// TwinCAT 3 PLC project TcGeodetic
// Title: TcGeodetic
// Company: Burks Engineering
// Author: Andrew Burks
// ProjectVersion: 0.2.3
// Description: Geodetic transformation library
// ProgramVersion: 3.1.4023.0
// libraries:
//   Tc2_Standard, * (Beckhoff Automation GmbH)
//   Tc2_System, * (Beckhoff Automation GmbH)
//   TcMatrix, * (Burks Engineering)
//   TcTransform, * (Burks Engineering)
// project tree:
//   GVLs/ GeoEllipsoids.TcGVL
//   POUs/ GeoEllipsoid.TcPOU, GeoPose.TcPOU, GeoPosition.TcPOU
//   Version/ Global_Version.TcGVL

// ---- GVLs/GeoEllipsoids.TcGVL
{attribute 'qualified_only'}
VAR_GLOBAL
	WGS84 : GeoEllipsoid('WGS-84', 6378137.0, 1.0 / 298.257223563);
	GRS80 : GeoEllipsoid('GRS-80', 6378137.0, 1.0 / 298.257222101);
	PZ90 :  GeoEllipsoid('PZ-90' , 6378136.0, 1.0 / 298.257839303);
END_VAR

// ---- Version/Global_Version.TcGVL
{attribute 'TcGenerated'}
{attribute 'no-analysis'}
{attribute 'linkalways'}
// This function has been automatically generated from the project information.
VAR_GLOBAL CONSTANT
	{attribute 'const_non_replaced'}
	stLibVersion_TcGeodetic : ST_LibVersion := (iMajor := 0, iMinor := 2, iBuild := 3, iRevision := 0, nFlags := 0, sVersion := '0.2.3');
END_VAR

// ---- POUs/GeoEllipsoid.TcPOU
(*
Geodetic Ellipsoid
----------------

Overview
================

Represents a geodetic reference ellipsoid (but not a geodetic datum). Contains functions for transitioning between latitude/longitude and XYZ coordinates.

To access standard ellipsoids use the GVL 'GeoEllipsoids'.	They cannot be copied, but you can use REFERENCE TO types to keep a shorthand copy somewhere.

.. note:: When creating an instance of this FB you *must* provide the name, semimajor axis, and flattening due to the use of FB_init parameters.
*)
{attribute 'no_assign'}
FUNCTION_BLOCK GeoEllipsoid
VAR_INPUT
END_VAR
VAR_OUTPUT
END_VAR
VAR
	Name_ : T_MaxString;
	SemiMajorAxis_ : LREAL;
	Flattening_ : LREAL;
END_VAR

METHOD FB_init : BOOL
VAR_INPUT
	bInitRetains : BOOL; // if TRUE, the retain variables are initialized (warm start / cold start)
	bInCopyCode : BOOL;  // if TRUE, the instance afterwards gets moved into the copy code (online change)
	
	eName : T_MaxString;
	eSemiMajorAxis : LREAL;//meters
	eFlattening : LREAL;//very small number
END_VAR
Name_ := eName;
SemiMajorAxis_ := eSemiMajorAxis;
Flattening_ := eFlattening;
END_METHOD

PROPERTY PUBLIC Flattening : LREAL
GET
Flattening := Flattening_;
END_GET
END_PROPERTY

METHOD PUBLIC GetCartesianFromGeodetic : Vector3
VAR_INPUT
	P : GeoPosition;
END_VAR
VAR
	N : LREAL;
END_VAR
N := GetNormalRadiusOfCurvature(P.LatitudeRad);

GetCartesianFromGeodetic.X := (N + P.Elevation) * COS(P.LatitudeRad) * COS(P.LongitudeRad);
GetCartesianFromGeodetic.Y := (N + P.Elevation) * COS(P.LatitudeRad) * SIN(P.LongitudeRad);
GetCartesianFromGeodetic.Z := ((1.0 - GetEccentricitySquared())*N + P.Elevation) * SIN(P.LatitudeRad);
END_METHOD

METHOD PROTECTED GetEccentricitySquared : LREAL
VAR_INPUT
END_VAR
GetEccentricitySquared := (2.0-Flattening)*Flattening;
END_METHOD

METHOD PROTECTED GetGeocentricLatitude : LREAL//radians
VAR_INPUT
	GeodeticLatitude : LREAL;//radians
END_VAR
GetGeocentricLatitude := ATAN((1-Flattening_) * (1-Flattening_)*TAN(GeodeticLatitude));
END_METHOD

METHOD PUBLIC GetGeodeticFromCartesian : GeoPosition
VAR_INPUT
	V : Vector3;
END_VAR
VAR
	RadLatitude_2 : LREAL;// 		'Q^2' 		from paper
	Magnitude_2 : LREAL;// 			'r^2' 		from paper
	Eccentricity_2 : LREAL;// 		'E^2' 		from paper
	AdjustedMag_2 : LREAL;// 		'r^2 - E^2' from paper
	SemiMinorConfocal_2 : LREAL;// 	'u^2' 		from paper
	SemiMajorConfocal_2 : LREAL;// 	'u^2' + E^2 from paper
	TanGeocentricLatitude : LREAL;// tan(beta) 	from paper
	GeocentricLatitude : LREAL;//   'beta' 		from paper
	AxialElevation : LREAL;
	RadialElevation : LREAL;
END_VAR
//stolen from : http://ir.lib.ncku.edu.tw/bitstream/987654321/39750/1/3011200501001.pdf
//error is <1mm for anything within 100km of the surface of the earth

RadLatitude_2 := V.X*V.X + V.Y*V.Y;
Magnitude_2 := RadLatitude_2 + V.Z* V.Z;

//right at pole longitude is indetermiante
IF RadLatitude_2 = 0 THEN
	GetGeodeticFromCartesian.LongitudeRad := 0;
ELSE
	GetGeodeticFromCartesian.LongitudeRad := atan2(V.Y,V.X);//eq 4c from paper
END_IF

//too close to poles for stuff to work well
IF RadLatitude_2 < (SemiMajorAxis * SemiMinorAxis * 1E-32) THEN
	//center of earth...angles dont even matter anymore
	IF V.Z = 0 THEN
		GetGeodeticFromCartesian.LatitudeRad := 0;
		GetGeodeticFromCartesian.Elevation := Magnitude_2;
	ELSE
		GetGeodeticFromCartesian.LatitudeRad := PI /2 * V.Z / ABS(V.Z);
		GetGeodeticFromCartesian.Elevation := ABS(V.Z) - SemiMinorAxis;
	END_IF;
ELSE
	Eccentricity_2 := SemiMajorAxis*SemiMajorAxis - SemiMinorAxis * SemiMinorAxis;
	AdjustedMag_2 := Magnitude_2 - Eccentricity_2;
	SemiMinorConfocal_2 := 0.5*AdjustedMag_2 + 0.5*SQRT(EXPT(AdjustedMag_2,2) + 4*Eccentricity_2*V.Z*V.Z); //eq 4a from paper
	SemiMajorConfocal_2 := SemiMinorConfocal_2 + Eccentricity_2;
	IF SQRT(SemiMinorConfocal_2) / SQRT(SemiMajorConfocal_2) < 10E-10 THEN
		//avoid divide by near zero when confocal is nearly flat and assumption of geocentric latidude equivalence atan(confocal) ~= atan(ellipsoid) stops being true
		IF V.Z = 0 THEN
			GeocentricLatitude := 0;
		ELSE
			GeocentricLatitude := PI/2 * V.Z/ABS(V.Z);
		END_IF;
		GetGeodeticFromCartesian.LatitudeRad := GeocentricLatitude;
	ELSE
		TanGeocentricLatitude := (SQRT(SemiMajorConfocal_2) * V.Z) / (SQRT(SemiMinorConfocal_2)*SQRT(RadLatitude_2));
		GeocentricLatitude := ATAN(TanGeocentricLatitude); //eq 6 from paper
		GetGeodeticFromCartesian.LatitudeRad := ATAN(SemiMajorAxis / SemiMinorAxis * TanGeocentricLatitude);
	END_IF;
	
	AxialElevation := V.Z - SemiMinorAxis*SIN(GeocentricLatitude);
	RadialElevation := SQRT(RadLatitude_2) - SemiMajorAxis*COS(GeocentricLatitude);
	
	GetGeodeticFromCartesian.Elevation := SQRT(AxialElevation*AxialElevation + RadialElevation*RadialElevation); //eq 7 from paper
	IF AxialElevation < 0 AND RadialElevation < 0 THEN
		GetGeodeticFromCartesian.Elevation := -1 * GetGeodeticFromCartesian.Elevation;
	END_IF

END_IF
END_METHOD

METHOD PROTECTED GetNormalRadiusOfCurvature : LREAL
VAR_INPUT
	lat : LREAL;//radians
END_VAR
VAR
	acosf : LREAL;
	bcosf : LREAL;
	den : LREAL;
END_VAR
acosf := SemiMajorAxis * COS(lat);
bcosf := GetSemiMinorAxis() * SIN(lat);
den := SQRT(acosf*acosf + bcosf*bcosf);
IF den = 0 THEN
	GetNormalRadiusOfCurvature := 0;
	ADSLOGSTR(ADSLOG_MSGTYPE_WARN,'GeodeticPosition::GetNormalRadiusOfCurvature Divide By Zero attempt in reference ellipsoid %s',Name);
	RETURN;
END_IF
GetNormalRadiusOfCurvature := SemiMajorAxis*SemiMajorAxis/den;
END_METHOD

METHOD PROTECTED GetSemiMinorAxis : LREAL
VAR_INPUT
END_VAR
GetSemiMinorAxis := SemiMajorAxis * (1-Flattening);
END_METHOD

METHOD PUBLIC GetTangentEnuRotation : RMatrix
VAR_INPUT
	P : GeoPosition;
END_VAR
VAR
	R_ENU : RMatrix;
	R_Lon : Rmatrix;
	R_Lat : Rmatrix;
	V : Vector3;
END_VAR
GetTangentEnuRotation := GetTangentXyuRotation(P,0.0);
RETURN;

//ECEF has X as 'up',   y as 'east',  Z as 'north' as lat=lon=0, translated to surface
//ENU  has X as 'east', y as 'north', z as 'up'
//therefore, the base rotation (ignoring lat/lon changes) should be: (projecting ENU unit vecotrs onto ECEF CS)
// [  0   0   1
//    1   0   0
//    0   1   0   ]

GetTangentEnuRotation.FillTrapezoidal(0,0,0);
GetTangentEnuRotation.SetRC(1,0,1);
GetTangentEnuRotation.SetRC(2,1,1);
GetTangentEnuRotation.SetRC(0,2,1);


R_Lon.SetFromAngle(P.LongitudeRad,Dimension.Z);//positive intrinsic rotation around ECEF Z
R_Lat.SetFromAngle(-1*P.LatitudeRad,Dimension.Y);//negative instrinsic rotation around rotated ECEF Y

GetTangentEnuRotation.RotateBy(R_Lat);
GetTangentEnuRotation.RotateBy(R_Lon);
END_METHOD

METHOD PUBLIC GetTangentEnuTransform : HMatrix
VAR_INPUT
	P : GeoPosition;
END_VAR
VAR
	R_ENU : RMatrix;
	R_Lon : Rmatrix;
	R_Lat : Rmatrix;
	V : Vector3;
END_VAR
V := GetCartesianFromGeodetic(P);
GetTangentEnuTransform.SetFromComponents(GetTangentEnuRotation(P),V);
END_METHOD

METHOD PUBLIC GetTangentXyuRotation : RMatrix
VAR_INPUT
	P : GeoPosition;
	Angle : LREAL;//radians of extra angle around the 'up' vector, from ENU
END_VAR
VAR
	R_ENU : RMatrix;
	R_Lon : Rmatrix;
	R_Lat : Rmatrix;
	RHeading : RMatrix;
	V : Vector3;
END_VAR
//ECEF has X as 'up',   y as 'east',  Z as 'north' as lat=lon=0, translated to surface
//ENU  has X as 'east', y as 'north', z as 'up'
//therefore, the base rotation (ignoring lat/lon changes) should be: (projecting ENU unit vecotrs onto ECEF CS)
// [  0   0   1
//    1   0   0
//    0   1   0   ]

GetTangentXyuRotation.SetFromAngle(Angle,Dimension.Z);

R_ENU.FillTrapezoidal(0,0,0);
R_ENU.SetRC(1,0,1);
R_ENU.SetRC(2,1,1);
R_ENU.SetRC(0,2,1);

R_Lon.SetFromAngle(P.LongitudeRad,Dimension.Z);//positive intrinsic rotation around ECEF Z
R_Lat.SetFromAngle(-1*P.LatitudeRad,Dimension.Y);//negative instrinsic rotation around rotated ECEF Y

GetTangentXyuRotation.RotateBy(R_ENU);
GetTangentXyuRotation.RotateBy(R_Lat);
GetTangentXyuRotation.RotateBy(R_Lon);
END_METHOD

METHOD PUBLIC GetTangentXyuTransform : HMatrix
VAR_INPUT
	P : GeoPosition;
	Angle : LREAL;//radians of extra normal rotation
END_VAR
VAR
	R_ENU : RMatrix;
	R_Lon : Rmatrix;
	R_Lat : Rmatrix;
	V : Vector3;
END_VAR
V := GetCartesianFromGeodetic(P);
GetTangentXyuTransform.SetFromComponents(GetTangentXyuRotation(P,Angle),V);
END_METHOD

PROPERTY PUBLIC Name : T_MaxString
GET
Name := Name_;
END_GET
END_PROPERTY

//meters
PROPERTY PUBLIC SemiMajorAxis : LREAL
GET
SemiMajorAxis := SemiMajorAxis_;
END_GET
END_PROPERTY

PROPERTY PUBLIC SemiMinorAxis : LREAL
GET
SemiMinorAxis := SemiMajorAxis*(1-Flattening);
END_GET
END_PROPERTY

END_FUNCTION_BLOCK

// ---- POUs/GeoPosition.TcPOU
(*
Geographic Position
----------------

Overview
================

Represents a geodetic (or geocentric) position with latitude, longitude, and elevation (above the ellipsoid).
*)
FUNCTION_BLOCK GeoPosition
VAR_INPUT
END_VAR
VAR_OUTPUT
END_VAR
VAR
	Latitude_  : LREAL;//radians north of equator
	Longitude_ : LREAL;//radians east of meridian
	Elevation_ : LREAL;//m above ellipsoid
END_VAR

METHOD PUBLIC Clear
VAR_INPUT
END_VAR
Latitude_ := 0;
Longitude_ := 0;
Elevation_ := 0;
END_METHOD

METHOD PUBLIC CopyFrom
VAR_INPUT
	P : GeoPosition;
END_VAR
Latitude_ := P.LatitudeRad;
Longitude_ := P.LongitudeRad;
Elevation_ := P.Elevation;
END_METHOD

PROPERTY PUBLIC Elevation : LREAL
GET
Elevation := Elevation_;
END_GET
SET
Elevation_ := Elevation;
END_SET
END_PROPERTY

METHOD PUBLIC GetCartesianPosition : Vector3
VAR_INPUT
	Ref : REFERENCE TO GeoEllipsoid := GeoEllipsoids.WGS84;
END_VAR
IF NOT(__ISVALIDREF(Ref)) THEN
	GetCartesianPosition := GeoEllipsoids.WGS84.GetCartesianFromGeodetic(THIS^);
ELSE
	GetCartesianPosition := Ref.GetCartesianFromGeodetic(THIS^);
END_IF;
END_METHOD

//Gets the relative position of the supplied GeoPosition, considering this GeoPosition as an ENU tangent reference frame
METHOD PUBLIC GetRelativePosition : Vector3
VAR_INPUT
	P : GeoPosition;
	Ref : REFERENCE TO GeoEllipsoid := GeoEllipsoids.WGS84;
END_VAR
VAR
	EnuInEcef : HMatrix;
END_VAR
EnuInEcef := GetTangentEnuTransform(Ref);
GetRelativePosition := EnuInEcef.GetTransformedVector3Reverse(P.GetCartesianPosition(Ref));
END_METHOD

METHOD PUBLIC GetTangentEnuPose : GeoPose
VAR_INPUT
	Ref : REFERENCE TO GeoEllipsoid := GeoEllipsoids.WGS84;
END_VAR
GetTangentEnuPose.SetFromEcefTransformation(GetTangentEnuTransform(Ref),Ref);
END_METHOD

METHOD PUBLIC GetTangentEnuRotation : RMatrix
VAR_INPUT
	Ref : REFERENCE TO GeoEllipsoid := GeoEllipsoids.WGS84;
END_VAR
IF NOT(__ISVALIDREF(Ref)) THEN
	GetTangentEnuRotation := GeoEllipsoids.WGS84.GetTangentEnurotation(THIS^);
ELSE
	GetTangentEnuRotation := Ref.GetTangentEnurotation(THIS^);
END_IF
END_METHOD

METHOD PUBLIC GetTangentEnuTransform : HMatrix
VAR_INPUT
	Ref : REFERENCE TO GeoEllipsoid := GeoEllipsoids.WGS84;
END_VAR
IF NOT(__ISVALIDREF(Ref)) THEN
	GetTangentEnuTransform := GeoEllipsoids.WGS84.GetTangentEnuTransform(THIS^);
ELSE
	GetTangentEnuTransform := Ref.GetTangentEnuTransform(THIS^);
END_IF
END_METHOD

METHOD PUBLIC IsEqual : BOOL
VAR_INPUT
	P : REFERENCE TO GeoPosition;
END_VAR
IsEqual := IsNearlyEqual(P,0.0,0.0);
END_METHOD

METHOD PUBLIC IsNearlyEqual : BOOL
VAR_INPUT
	P : REFERENCE TO GeoPosition;
	PrecisionLatLon : LREAL;//radians
	PrecisionElevation : LREAL;//meters
END_VAR
IsNearlyEqual := ABS(P.LatitudeRad 		- LatitudeRad) 	<= PrecisionLatLon
             AND ABS(P.LongitudeRad 	- LongitudeRad) <= PrecisionLatLon
             AND ABS(P.Elevation 		- Elevation)	<= PrecisionElevation;
END_METHOD

PROPERTY PUBLIC LatitudeDeg : LREAL
GET
LatitudeDeg := 180.0 * Latitude_ /PI;
END_GET
SET
Latitude_ := PI * LatitudeDeg / 180.0;
END_SET
END_PROPERTY

PROPERTY PUBLIC LatitudeRad : LREAL
GET
LatitudeRad := Latitude_;
END_GET
SET
Latitude_ := LatitudeRad;
END_SET
END_PROPERTY

PROPERTY PUBLIC LongitudeDeg : LREAL
GET
LongitudeDeg := 180.0 * Longitude_ /PI;
END_GET
SET
Longitude_ := PI * LongitudeDeg / 180.0;
END_SET
END_PROPERTY

PROPERTY PUBLIC LongitudeRad : LREAL
GET
LongitudeRad := Longitude_;
END_GET
SET
Longitude_ := LongitudeRad;
END_SET
END_PROPERTY

METHOD PUBLIC SetFromCartesianPosition
VAR_INPUT
	V : Vector3;
	Ref : REFERENCE TO GeoEllipsoid;
END_VAR
VAR
	P : GeoPosition;
END_VAR
IF NOT(__ISVALIDREF(Ref)) THEN
	P := GeoEllipsoids.WGS84.GetGeodeticFromCartesian(V);
ELSE
	P := Ref.GetGeodeticFromCartesian(V);
END_IF
CopyFrom(P);
END_METHOD

METHOD PUBLIC SetFromComponentsDeg
VAR_INPUT
	Lat : LREAL;
	Lon : LREAL;
	El : LREAL;
END_VAR
LatitudeDeg := Lat;
LongitudeDeg := Lon;
Elevation := El;
END_METHOD

METHOD PUBLIC SetFromComponentsRad
VAR_INPUT
	Lat : LREAL;
	Lon : LREAL;
	El : LREAL;
END_VAR
LatitudeRad := Lat;
LongitudeRad := Lon;
Elevation := El;
END_METHOD

END_FUNCTION_BLOCK

// ---- POUs/GeoPose.TcPOU
(*
Geographic Pose
----------------

Overview
================
Represents a coordinate system on a reference ellipsoid.
Similar to the HMatrix transformation, but based on an ellipsoid instead of in cartesian space (helper functions are included to switch between HMatrix and GeoPose).
Represents the geodetic (or geocentric) position with latitude, longitude, and elevation (above the ellipsoid) - Accessed with the 'Position' property.
Represents the orientation as a set of angles relative to the ENU tangent coordinate system at the CS origin - Accessed with the 'Orientation' property.
*)
FUNCTION_BLOCK GeoPose
VAR_INPUT
END_VAR
VAR_OUTPUT
END_VAR
VAR
	Position_ : GeoPosition;//ECEF
	Orientation_ : TaitBryanAngleOrientation;//ENU at position
END_VAR

METHOD PUBLIC Clear
VAR_INPUT
END_VAR
Position_.Clear();
Orientation_.Clear();
END_METHOD

METHOD PUBLIC CopyFrom
VAR_INPUT
	P : GeoPose;
END_VAR
Position_.CopyFrom(P.Position_);
Orientation_.CopyFrom(P.Orientation_);
END_METHOD

METHOD PUBLIC GetEcefTransformation : HMatrix
VAR_INPUT
	Ref : REFERENCE TO GeoEllipsoid := GeoEllipsoids.WGS84;
END_VAR
VAR
	EnuInEcef : HMatrix;//holds the geoposition part, and the tangent rotation
	ThisInEnu : HMatrix;//just holds the local rotation portion
END_VAR
EnuInEcef := Position_.GetTangentEnuTransform(Ref);
ThisInEnu.RMatrixComponent := Orientation_.GetRMatrix();
GetEcefTransformation := EnuInEcef.GetTransformedHMatrix(ThisInEnu);
END_METHOD

METHOD PUBLIC GetRelativeOrientation : TaitBryanAngleOrientation
VAR_INPUT
	P : GeoPose;
	Ref : REFERENCE TO GeoEllipsoid := GeoEllipsoids.WGS84;
END_VAR
VAR
	ThisInEcef : HMatrix;
	InputInThis : HMatrix;
END_VAR
ThisInEcef := GetEcefTransformation(Ref);
InputInThis := ThisInEcef.GetTransformedHMatrixReverse(P.GetEcefTransformation(Ref));
GetRelativeOrientation.SetFromRMatrix(InputInThis.RMatrixComponent);
END_METHOD

METHOD PUBLIC GetRelativePosition : Vector3
VAR_INPUT
	P : GeoPose;
	Ref : REFERENCE TO GeoEllipsoid := GeoEllipsoids.WGS84;
END_VAR
VAR
	ThisInEcef : HMatrix;
	InputInThis : HMatrix;
END_VAR
ThisInEcef := GetEcefTransformation(Ref);
InputInThis := ThisInEcef.GetTransformedHMatrixReverse(P.GetEcefTransformation(Ref));
GetRelativePosition := InputInThis.Vector3Component;
END_METHOD

METHOD PUBLIC IsEqual : BOOL
VAR_INPUT
	P : GeoPose;
END_VAR
IsEqual := IsNearlyEqual(P,0.0,0.0,0.0);
END_METHOD

METHOD PUBLIC IsNearlyEqual : BOOL
VAR_INPUT
	P : GeoPose;
	PositionPrecisionLatLon : LREAL;//rad
	PositionPrecisionElevation : LREAL;//m
	OrientationPrecision : LREAL;//radians
END_VAR
IsNearlyEqual := Position_.IsNearlyEqual(P.Position_, PositionPrecisionLatLon, PositionPrecisionElevation) AND Orientation_.IsNearlyEqual(P.Orientation_, OrientationPrecision);
END_METHOD

PROPERTY PUBLIC Orientation : TaitBryanAngleOrientation
GET
Orientation.CopyFrom(Orientation_);
END_GET
SET
Orientation_.CopyFrom(Orientation);
END_SET
END_PROPERTY

PROPERTY PUBLIC Position : GeoPosition
GET
Position.CopyFrom(Position_);
END_GET
SET
Position_.CopyFrom(Position);
END_SET
END_PROPERTY

METHOD PUBLIC SetFromComponents
VAR_INPUT
	P : GeoPosition;
	O : TaitBryanAngleOrientation;
END_VAR
Position_.CopyFrom(P);
Orientation_.CopyFrom(O);
END_METHOD

METHOD PUBLIC SetFromEcefTransformation
VAR_INPUT
	H : HMatrix;//ThisInEcef)
	Ref : REFERENCE TO GeoEllipsoid := GeoEllipsoids.WGS84;
END_VAR
VAR
	EnuInEcef : HMatrix;
	ThisInEnu : HMatrix;
END_VAR
Clear();
Position_.SetFromCartesianPosition(H.Vector3Component,Ref);
EnuInEcef := Position_.GetTangentEnuTransform(Ref);
ThisInEnu := EnuInEcef.GetTransformedHMatrixReverse(H);
Orientation_.SetFromRMatrix(ThisInEnu.RMatrixComponent);
END_METHOD

END_FUNCTION_BLOCK
